# EPICS substitutions: db/MicroEpsilon/ecmcOptoILD2300_50mm.substitutions
file "ecmcOptoILD2300_XXmm_chX.template"
{
  pattern {CH_ID, LINR,     ESLO,     EOFF,   EGU,     PREC }
          {01,    "SLOPE",  1e-6,     0,      "mm",    5    }
}
